PROGRAM Running_Sequence
VAR
	zz_EP : INT; 
	Cognex_IS7K_01: FB_CameraControl;
END_VAR

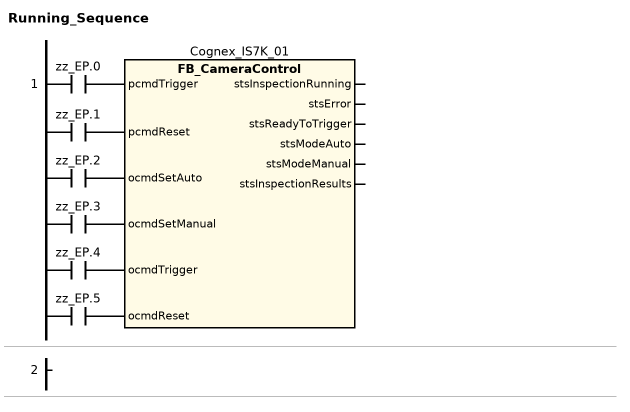
// NETWORK 1
Cognex_IS7K_01(
    pcmdTrigger := zz_EP.0,
    pcmdReset := zz_EP.1,
    ocmdSetAuto := zz_EP.2,
    ocmdSetManual := zz_EP.3,
    ocmdTrigger := zz_EP.4,
    ocmdReset := zz_EP.5); // FB_CameraControl

// NETWORK 2

END_PROGRAM

(* stored: Version 1.1.0.1, ProductVersion 3.1.4024.13
   POU Running_Sequence: Id {b9bea037-5906-405f-b72d-3d1d48ae1070}, SpecialFunc None *)
